FUNCTION_BLOCK xscal_f
VAR_INPUT
    b_n: DINT;
    a: LREAL;
    ix0: DINT;
END_VAR
VAR_IN_OUT
    x: ARRAY [0..4] OF LREAL;
END_VAR
VAR_TEMP
    b: DINT;
    k: DINT;
END_VAR

b := (ix0 + b_n) - 1;
k := ix0;
WHILE k <= b DO
    x[k - 1] := x[k - 1] * a;
    k := k + 1;
END_WHILE;

END_FUNCTION_BLOCK

(* stored: Version 1.1.0.1, ProductVersion 3.1.4024.12
   POU xscal_f: Id {1186c4ef-f42c-4054-b819-9da7e5ff668e}, SpecialFunc None *)
